// TwinCAT 3 PLC project Alles_Samen
// ProgramVersion: 3.1.4022.1
// libraries:
//   Tc2_Standard, * (Beckhoff Automation GmbH)
//   Tc2_System, * (Beckhoff Automation GmbH)
//   Tc2_TcpIp, * (Beckhoff Automation GmbH)
//   Tc2_Utilities, * (Beckhoff Automation GmbH)
//   Tc3_JsonXml, * (Beckhoff Automation GmbH)
//   Tc3_Module, * (Beckhoff Automation GmbH)
//   ERS_CO2 Payload Decoder,1.0,PXL-Tech
//   MSC1608 Payload Decoder,1.0,PXL-Tech
// project tree:
//   DUTs/ ST_Gwrx.TcDUT, ST_MoteTx.TcDUT, ST_UserData.TcDUT
//   / GlobalTextList.TcGTLO, PlcTask.TcTTO, Visualization Manager.TcVMO (not stored)
//   GVLs/ GVL_1.TcGVL
//   POUs/ Decoder.TcPOU, DecoderCO2.TcPOU, Json_XML.TcPOU, MAIN.TcPOU, Tcp_ip.TcPOU
//   VISUs/ Visualization_1.TcVIS
// real-time tasks:
//   TASK PlcTask: cycle T#10ms, priority 20, ADS port 350

CONFIGURATION Alles_Samen
    RESOURCE PLC ON TwinCAT3
        TASK PlcTask(INTERVAL := T#10ms, PRIORITY := 20);
        PROGRAM MAIN WITH PlcTask : MAIN;
    END_RESOURCE
END_CONFIGURATION

// ---- DUTs/ST_Gwrx.TcDUT
TYPE ST_Gwrx :
STRUCT
	TimeRec	: STRING;//DATE_AND_TIME ;
	Chan : DINT ;
	Rfch : DINT ;
	Rssi : DINT ;
	Lsnr : REAL ;
END_STRUCT
END_TYPE

// ---- DUTs/ST_MoteTx.TcDUT
TYPE ST_MoteTx :
STRUCT
	Freq	: DINT ;
	Modu	: STRING(20);
	Datr	: STRING(20);
	Codr	: STRING(20);
END_STRUCT
END_TYPE

// ---- DUTs/ST_UserData.TcDUT
TYPE ST_UserData :
STRUCT
	SeqNo	: DINT;
	Port	: DINT;
	Payload	: STRING;
	Payload2: DINT;
	MoteTx	: ST_MoteTx;
	Gwrx : ST_Gwrx;
END_STRUCT
END_TYPE

// ---- GVLs/GVL_1.TcGVL
VAR_GLOBAL
	sDatastring: STRING(500);
	
	Moteeui			: STRING;
	Appeui			: STRING;
	UserData		: ST_UserData;
	PayloadDecoded	: STRING;

	PayloadLength	: DINT;
	PayloadData		: ARRAY[1..100] OF BYTE;
	NullByte		: BYTE := 0;

END_VAR

// ---- POUs/MAIN.TcPOU
PROGRAM MAIN
VAR
END_VAR

Tcp_ip();

END_PROGRAM

// ---- POUs/Tcp_ip.TcPOU
PROGRAM Tcp_ip
VAR
	bConnect: BOOL;
	bRecieve: BOOL;
	FB_create: FB_SocketUdpCreate;
	FB_Recieve: FB_SocketUdpReceiveFrom;
	FB_close: FB_SocketClose;
	data : ARRAY[0..500] OF BYTE;
END_VAR

FB_create(
	sSrvNetId:= , 							//Lokaal netwerk (mag leeg blijven)
	sLocalHost:= '192.168.1.82', 			//Eigen ip van de PC en ingesteld in de gateway gekregen van Dieter
	nLocalPort:= 811,						//Ingesteld op de gateway
	bExecute:= bConnect,					//Trigger voor functieblok
	tTimeout:= T#1S);
	

FB_Recieve(
	sSrvNetId:= , 									//Lokaal netwerk (mag leeg blijven)
	hSocket:= FB_create.hSocket,					 
	cbLen:= SIZEOF(data), 							//Kijkt naar de lengte van het bericht
	pDest:= ADR(data), 								//Plaat waar de het bericht wordt opgeslaan
	bExecute:= NOT FB_recieve.bBusy AND bRecieve, 	//Trigger voor functieblok
	tTimeout:= T#1S);
	
FB_close(
	sSrvNetId:= , 							//Lokaal netwerk (mag leeg blijven)
	hSocket:= FB_create.hSocket, 			
	bExecute:= NOT bConnect, 				//Sluiten van de connectie 
	tTimeout:= T#1S);
	
IF FB_Recieve.nRecBytes > 0 THEN 										//Dit gebuert op het moment dat er data binnenkomt
	memcpy(ADR(sDatastring),ADR(data),FB_Recieve.nRecBytes);			//Het bericht zal worden opgeslaan in Datastring
	memcpy(ADR(sDatastring) + FB_Recieve.nRecBytes,ADR(NullByte),1);	//Nullbyte word gedetecteerd stoppen met bericht plaatsen
	Json_XML();															//Oproepen POU Json_XML - MOET hier anders bluescreen
	Decoder();
	DecoderCO2();															//Oproepen POU Decoder  - MOET hier anders bluescreen
END_IF

END_PROGRAM

// ---- POUs/Json_XML.TcPOU
PROGRAM Json_XML
VAR
	
	//sJsontest		: STRING(500) := '{"rx": {"moteeui": "00-59-ac-00-00-15-10-ee", "appeui": "0000000000000000", "userdata": {"seqno": 122, "port": 1, "payload": "MDIwMDA1YWUwOTdhMzYwMDAwZmEwMDAwMDAwMDAwMDA=", "motetx": {"freq": 868300000, "modu": "LoRa", "datr": "SF8BW125", "codr": "4/5"}}, "gwrx":  [{"time": "2017-10-17 12:34:53", "chan": 4, "rfch": 0, "rssi": -34, "lsnr": 11.800000000000001}]}}';	
	//sJsontest		: STRING(500) := '{"rx": {"moteeui": "00-59-ac-00-00-15-10-ee", "appeui": "0000000000000000", "userdata": {"seqno": 122, "port": 1, "payload": "MDIwMDA1YWUwOTdhMzYwMDAwZmEwMDAwMDAwMDAwMDA=", "motetx": {"freq": 868300000, "modu": "LoRa", "datr": "SF8BW125", "codr": "4/5"}}, "gwrx": [{"time": "2017-10-17 12:34:53", "chan": 4, "rfch": 0, "rssi": -34, "lsnr": 11.800000000000001}]}}';	
	
	x : DINT;
	g : STRING;
	fbJson			: FB_JsonDomParser;
	JsonDoc			: SJsonValue;
	Json_St1		: SJsonValue;
	JSon_St2		: SJsonValue; 
	JSon_St3		: SJsonValue;
	JSon_St4		: SJsonValue;
	JSon_St5		: SJsonValue;
	JSon_St6		: SJsonValue;
	Stringdata		: STRING;
	
	i: INT;
END_VAR

FOR i := 0 TO 498 DO										//Forloop doorloop elk teken appart
	IF sDatastring[i] = 91 OR sDatastring[i] = 93 THEN		//ALs er een vierkante haak  voor komt
		sDatastring[i] := 32;								//Zal het door een spatie gewijzigd worden
	END_IF
END_FOR
 
JsonDoc := fbJson.ParseDocument(sDatastring);

// rx
Json_St1 := fbJson.FindMember(jsonDoc, 'rx');			

	// moteeui 
	JSon_St2 := fbJson.FindMember(Json_St1, 'moteeui');
	Moteeui := fbJson.GetString(JSon_St2);

	// appeui	
	JSon_St2 := fbJson.FindMember(Json_St1, 'appeui');
	Appeui := fbJson.GetString(JSon_St2);

	// userdata
	JSon_St2 := fbJson.FindMember(Json_St1, 'userdata');

		// seqno
		JSon_St3 := fbJson.FindMember(Json_St2, 'seqno');
		UserData.SeqNo := fbJson.GetInt(JSon_St3);

		// port
		JSon_St3 := fbJson.FindMember(Json_St2, 'port');
		UserData.Port := fbJson.GetInt(JSon_St3);

		// payload
		JSon_St3 := fbJson.FindMember(Json_St2, 'payload');
		UserData.Payload := fbJson.GetString(JSon_St3);
		PayloadLength:= fbJson.GetBase64(JSon_St3, ADR(PayloadData), SIZEOF(PayloadData));
		Memcpy(ADR(PayloadDecoded), ADR(PayloadData), PayloadLength);
		Memcpy(ADR(PayloadDecoded)+PayloadLength, adr(NullByte), 1);

		// motetx
		JSon_St3 := fbJson.FindMember(Json_St2, 'motetx');

			// freq
			JSon_St4 := fbJson.FindMember(Json_St3, 'freq');
			UserData.MoteTx.Freq := fbJson.GetInt(JSon_St4);

			// modu
			JSon_St4 := fbJson.FindMember(Json_St3, 'modu');
			UserData.MoteTx.Modu := fbJson.GetString(JSon_St4);

			// datr
			JSon_St4 := fbJson.FindMember(Json_St3, 'datr');
			UserData.MoteTx.Datr := fbJson.GetString(JSon_St4);

			// codr
			JSon_St4 := fbJson.FindMember(Json_St3, 'codr');
			UserData.MoteTx.Codr := fbJson.GetString(JSon_St4);

		// gwrx
		JSon_St5 := fbJson.FindMember(Json_St1, 'gwrx');
		Stringdata := fbJson.GetString(JSon_St5);

		// seqno
		JSon_St6 := fbJson.FindMember(Json_St5, 'time');
		UserData.gwrx.TimeRec  := fbJson.GetString(JSon_St6);

END_PROGRAM

// ---- POUs/Decoder.TcPOU
PROGRAM Decoder
VAR
 	FB_Decoder : MCS1608_Payload_Decoder;
    //GenSens
 	Status     			:BYTE;      // Content Depends on Message ID == for future use
	BaromBar			:REAL;      // Air Pressure in mBar
	Temp1   			:REAL;     	// in 0,01 degC
	Humidity   			:BYTE;      // Relative Humidity in %
	LevelX     			:SINT;      // Inverse Sinus of Spirit Level in Deg X-Direction -128 = -90 Degr .. +127 = +90 Degr
	LevelY     			:SINT;      // Inverse Sinus of Spirit Level in Deg Y-Direction -128 = -90 Degr .. +127 = +90 Degr
	LevelZ     			:SINT;      // Inverse Sinus of Spirit Level in Deg Z-Direction -128 = -90 Degr .. +127 = +90 Degr
	VibAmp     			:USINT;     // Amplitude of Vibration Detected == Future
	VibFreq    			:USINT;     // Approx. Frequency of Vibration Detected in Hz == Future



	//Tracking
	Start				:BOOL;// Start Message
	Moving				:BOOL;// Object Moving
	Stop				:BOOL;// Object Stopped
	Vibr				:BOOL;// Vibration Detected
	Temp2				:REAL;// Temperature in 0,01 degC
	GPSFixAge			:BYTE;// bit 0..7 = Age of last GPS Fix in Minutes,
	SatCnt_HiLL			:BYTE;// bit 0..4 = SatInFix, bit5 Latitude 25 bit 6,7 = Longitude 25,26
	Lat					:REAL;
	Lon					:REAL;
	
	//Alarm
	GravRotAl		:BOOL;	// Gravity Rotation Detected
	MagRot			:BOOL;	// Magnetic Rotation Detected
	MotAlarm		:BOOL;	// Motion Alarm Detected
	GeoFenceAl		:BOOL;	// GeoFence Violation Detected
	VibrAl			:BOOL;	// Vibration Alarm Detected
	ShockAl			:BOOL;	// Shock Alarm (future use)
	DigIn1Al		:BOOL;	// Digin1 Alarm Detected
	DigIn2Al		:BOOL;	// Digin2 Alarm Detected
	Temp			:REAL;	// Temperature in 0,01 Celcius
	Hum				:BYTE;	// Relative Humidity in %
	BaromBar2		:REAL;	// Air Pressure in Mbar
	
	Alarm1 : Alarm; 
END_VAR

FB_Decoder(dataString := PayloadDecoded);
 
CASE FB_Decoder.MsgID OF 
	FB_Decoder.ID_Tracking:
		//Start := FB_Decoder.Tracking.Start;
		Moving := FB_Decoder.Tracking.Moving;
		Stop := FB_Decoder.Tracking.Stop;
		Vibr := FB_Decoder.Tracking.Vibr;
		Temp2 := FB_Decoder.Tracking.Temp;
		GPSFixAge := FB_Decoder.Tracking.GPSFixAge;
		SatCnt_HiLL	:= FB_Decoder.Tracking.SatCnt_HiLL;
		Lat	:= FB_Decoder.Tracking.Lat;
		Lon	:= FB_Decoder.Tracking.Lon;
	FB_Decoder.ID_Alarm:
		Alarm1.MotAlarm := FB_Decoder.Alarm.MotAlarm;
	FB_Decoder.ID_GenSens:
		Status := FB_Decoder.GenSens.Status;
		BaromBar := FB_Decoder.GenSens.BaromBar;
		Temp := FB_Decoder.GenSens.Temp;
		Humidity := FB_Decoder.GenSens.Humidity;
		LevelX := FB_Decoder.GenSens.LevelX;
		LevelY := FB_Decoder.GenSens.LevelY;
		LevelZ := FB_Decoder.GenSens.LevelZ;
		VibAmp := FB_Decoder.GenSens.VibAmp;
		VibFreq := FB_Decoder.GenSens.VibFreq;
END_CASE

END_PROGRAM

// ---- POUs/DecoderCO2.TcPOU
PROGRAM DecoderCO2
VAR
	FB_Decoder : ERS_CO2_PayloadDecoder;
	
	Temperature 	: REAL;		//Temp -3276.8°C - 3276.7°C
	Humidity 		: BYTE;		//Humidity 0-100%
	X 				: REAL;		//Acceleration X -128 --> 127 +/-63 = 1G
	Y 				: REAL;		//Acceleration Y -128 --> 127 +/-63 = 1G
	Z 				: REAL;		//Acceleration Z -128 --> 127 +/-63 = 1G
	Light 			: WORD; 	//Light 0 - 65535 Lux
	Motion 			: BYTE;		//No of motion 0-255
	Co2				: WORD;		//Co2 0-65535 ppm 
	Vdd				: WORD;		//VDD 0-65535mV
	Analog1			: WORD;		//VDD 0-65535mV
	Lat				: DWORD;	//Latitude binary
	Lon				: DWORD;	//Longitude binary
	Pulse1			: WORD;		//Relative pulse count
	pulseAbs		: DWORD;	//no 0 - 0xFFFFFFFF
	ExternalTemp	: REAL;		//External temp -3276.5C-->3276.5C
	Digital			: BYTE;		//Value 1 or 0
	Distance		: WORD;		//Distance in mm
	AccMotion		: BYTE;		//Number of vibration/motion
	IrInternalTemp	: REAL;		//Internal temp -3276.5C - 3276.5C
	IrExternalTemp	: REAL;		//External temp -3276.5C - 3276.5C
	Occupancy		: BYTE;		//Data
	Waterleak		: BYTE;		//Data 0-255
	Pressure		: REAL;		//Pressure data(hPa)
	SoundPeak		: BYTE;		//Sound peak
	SoundAvg		: BYTE;		//Sound average
	Pulse2			: WORD;		//0 - 0xFFFF
	PulseAbs2		: DWORD;	//no 0 - 0xFFFFFFFF
	Analog2			: WORD;		//Voltage in mV
	ExternalTemp2	: REAL;		//External temp2 -3276.5C - 3276.5C
END_VAR

FB_Decoder(dataString := PayloadDecoded);
 
		Temperature 	:= FB_Decoder.Temperature;
		Humidity 		:= FB_Decoder.Humidity;
		X 				:= FB_Decoder.X;
		Y 				:= FB_Decoder.Y;
		Z 				:= FB_Decoder.Z;
		Light 			:= FB_Decoder.Light;		
		Motion 			:= FB_Decoder.Motion;
		Co2				:= FB_Decoder.Co2; 
		Vdd				:= FB_Decoder.Vdd;
		Analog1			:= FB_Decoder.Analog1;
		Lat				:= FB_Decoder.Lat;
		Lon				:= FB_Decoder.Lon;
		Pulse1			:= FB_Decoder.Pulse1;
		pulseAbs		:= FB_Decoder.pulseAbs;
		ExternalTemp	:= FB_Decoder.ExternalTemp;
		Digital			:= FB_Decoder.Digital;
		Distance		:= FB_Decoder.Distance;
		AccMotion		:= FB_Decoder.AccMotion;
		IrInternalTemp	:= FB_Decoder.IrInternalTemp;
		IrExternalTemp	:= FB_Decoder.IrExternalTemp;
		Occupancy		:= FB_Decoder.Occupancy;
		Waterleak		:= FB_Decoder.Waterleak;
		Pressure		:= FB_Decoder.Pressure;
		SoundPeak		:= FB_Decoder.SoundPeak;
		SoundAvg		:= FB_Decoder.SoundAvg;
		Pulse2			:= FB_Decoder.Pulse2;
		PulseAbs2		:= FB_Decoder.PulseAbs2;
		Analog2			:= FB_Decoder.Analog2;
		ExternalTemp2	:= FB_Decoder.ExternalTemp2;

END_PROGRAM

// ---- GlobalTextList.TcGTLO
TEXTLIST GlobalTextList
  370 = 'Bar : %d'
  367 = 'Close'
  732 = 'Conection'
  364 = 'Connect'
  731 = 'Create'
  677 = 'Datum/Tijd : '
  126 = 'Datum/Tijd : %s'
  729 = 'Error'
  723 = 'Humidity : %d %'
  724 = 'Level x : %d'
  725 = 'Level y : %d'
  726 = 'Level z : %d'
  368 = 'Mesage ID : %d'
  366 = 'Payload : %s'
  365 = 'Recieve'
  730 = 'Sensor ID : %s'
  369 = 'Status : %d'
  283 = 'Temp : %.2f °c'
  810 = 'Temp : %f °c'
  232 = 'Temp : %f.2 °c'
  371 = 'Temp : %i °c'
  66 = 'Temp : %r °c'
  733 = 'Type sensor : '
  727 = 'VibAmp : %d'
  728 = 'VidFreq : %d'
END_TEXTLIST

// ---- VISUs/Visualization_1.TcVIS
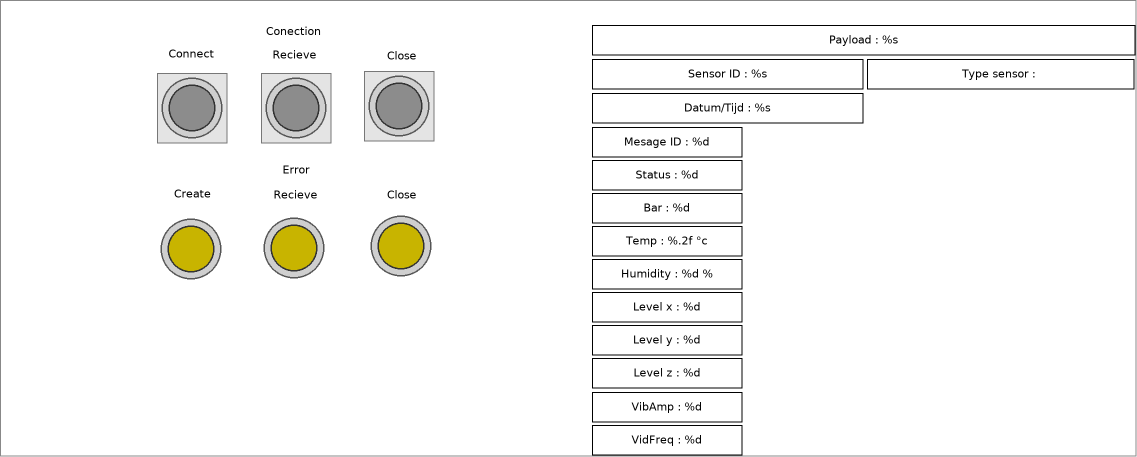
VISUALIZATION Visualization_1  // 1137x457
    PushSwitch (157,73 70x70), variable: Tcp_ip.bConnect, behaviour: TOGGLE, style: Switch-PushSwitch-Gray
    Label (156,39 71x30), "Connect"
    PushSwitch (261,73 70x70), variable: Tcp_ip.bRecieve, behaviour: TOGGLE, style: Switch-PushSwitch-Gray
    Label (261,40 67x30), "Recieve"
    Rectangle (592,25 543x30), "Payload : %s", text variable: PayloadDecoded
    PushSwitch (364,71 70x70), variable: Tcp_ip.FB_close.bExecute, behaviour: TOGGLE, style: Switch-PushSwitch-Gray
    Label (369,41 66x30), "Close"
    Rectangle (592,127 150x30), "Mesage ID : %d", text variable: Decoder.FB_Decoder.MsgID
    Rectangle (592,160 150x30), "Status : %d", text variable: Decoder.Status
    Rectangle (592,193 150x30), "Bar : %d", text variable: Decoder.BaromBar
    Rectangle (592,226 150x30), "Temp : %.2f °c", text variable: Decoder.Temp
    Rectangle (592,259 150x30), "Humidity : %d %", text variable: Decoder.Humidity
    Rectangle (592,292 150x30), "Level x : %d", text variable: Decoder.LevelX
    Rectangle (592,325 150x30), "Level y : %d", text variable: Decoder.LevelY
    Rectangle (592,358 150x30), "Level z : %d", text variable: Decoder.LevelZ
    Rectangle (592,392 150x30), "VibAmp : %d", text variable: Decoder.VibAmp
    Rectangle (592,425 150x30), "VidFreq : %d", text variable: Decoder.VibFreq
    Lamp1 (259,213 70x70), variable: Tcp_ip.FB_Recieve.bError, style: Lamp-Lamp1-Yellow
    Lamp1 (366,211 70x70), variable: Tcp_ip.FB_close.bError, style: Lamp-Lamp1-Yellow
    Lamp1 (156,214 70x70), variable: Tcp_ip.FB_create.bError, style: Lamp-Lamp1-Yellow
    Label (156,155 280x30), "Error"
    Rectangle (592,59 271x30), "Sensor ID : %s", text variable: Moteeui
    Label (157,179 71x30), "Create"
    Label (262,180 67x30), "Recieve"
    Label (369,180 66x30), "Close"
    Label (165,17 257x29), "Conection"
    Rectangle (867,59 267x30), "Type sensor :"
    Rectangle (592,93 271x30), "Datum/Tijd : %s", text variable: UserData.Gwrx.TimeRec
END_VISUALIZATION
